{attribute addProperty BoxType "KL6551"}
{attribute addProperty Id "Channel_1Channel_D70D803000"}
{attribute addProperty CRC "2063095037"}
{attribute addProperty SizeInBites "0"}
{attribute addProperty SizeInBytes "0"}
TYPE KL6551_7AF854FD :
STRUCT
	{attribute addProperty Name "Channel_1"}
	Channel_1 : Channel_D70D8030;
END_STRUCT
END_TYPE

(* stored: Version 1.2.0.0, ProductVersion 3.1.4024.9
   DUT KL6551_7AF854FD: Id {fa15af1e-8774-4c28-85cc-fcc2a426316c} *)
